(* CODESYS project CintasSoplado.project
   Title: CintasSoplado
   Version: 0.0.0.0
   Author: serbogr1

Project tree, tasks and I/O mapping:
  MyController : TM241CE40R, Schneider Electric, order no. TM241CE40R, version 4.0.6.18
    application Application
      libraries: Toolbox, 2.2.0.0 (Schneider Electric)
      task MAST (cyclic, interval 50 ms, priority 15, watchdog 100 ms x 1) calls ProcesoUno, ProcesoDos, Pulsadores, PID
      global variables GVL
      visualisation HMIW_Control
      image pool ImagePool
      program ProcesoDos [SFC]: E2_active, E8_active
      program ProcesoUno [SFC]: E8_active, E7_active, E9_active, E10_active, E11_active, E12_active
      program Pulsadores [LD]
      program PruebaAnalogica [ST]
      program PID [LD]
    DI : Digital Inputs, Schneider Electric, version 4.0.6.18
        input  idwDI_IDW0 : DWORD  // IDW0
        input  ibDI_IB1 : BYTE  // IB1
    DQ : Digital Outputs, Schneider Electric, version 4.0.6.18
        output qwDQ_QW0 : WORD  // QW0
        output qbDQ_QB1 : BYTE  // QB1
    Counters : Counters, Schneider Electric, version 4.0.6.18
    Pulse_Generators : Pulse Generators, Schneider Electric, version 4.0.6.18
    Cartridge_1 : Cartridge, Schneider Electric, version 4.0.6.18
      TMC4AI2 : TMC4AI2, Schneider Electric, order no. TMC4AI2, version 1.0.1.0
          input  iiTMC4AI2_IW0 : INT  // IW0
          input  iiTMC4AI2_IW1 : INT  // IW1
          input  ibTMC4AI2_IW2 : BYTE  // IW2
    Cartridge_2 : Cartridge, Schneider Electric, version 4.0.6.18
      TMC4AQ2 : TMC4AQ2, Schneider Electric, order no. TMC4AQ2, version 1.0.1.1
          output qiTMC4AQ2_QW0 : INT  // QW0
          output qiTMC4AQ2_QW1 : INT  // QW1
          input  ibTMC4AQ2_IW0 : BYTE  // IW0
    IO_Bus : IO bus - TM3, Schneider Electric, version 4.0.6.18
    COM_Bus : COM bus, Schneider Electric, version 4.0.6.18
    Ethernet_1 : Ethernet Network, Schneider Electric, version 4.0.6.18
        settings: WebServer = TRUE; FTP Server = TRUE; SoMachine Protocol = TRUE; Modbus Server = TRUE; NetManage Protocol = TRUE; SNMP protocol = TRUE; Enable Routing = FALSE; WebVisu protocol = TRUE; DHCP Server Active = FALSE
    Serial_Line_1 : Serial line, Schneider Electric, version 4.0.6.18
      SoMachine_Network_Manager : SoMachine-Network Manager, Schneider Electric, version 4.0.0.2
    Serial_Line_2 : Serial line, Schneider Electric, version 4.0.6.18
      Modbus_Manager : Modbus Manager, Schneider Electric, version 4.0.0.2
  text list GlobalTextList
*)

// MyController/Application/GVL
VAR_GLOBAL
END_VAR

// MyController/Application/ProcesoUno
PROGRAM ProcesoUno
VAR
	bS_FC_Empujador_1          AT %IX0.0: BOOL; (*I1*)
	bS_IC_Empujador_1          AT %IX0.1: BOOL; (*I2*)
	bS_FC_Empujador_2          AT %IX0.2: BOOL; (*I3*)
	bS_IC_Empujador_2          AT %IX0.3: BOOL; (*I4*)
	bS_FT_Empujador_1          AT %IX0.4: BOOL; (*I5*)
	bS_FT_Fresadora            AT %IX0.5: BOOL; (*I6*)
	bS_FT_Carga                AT %IX0.6: BOOL; (*I7*)
	bS_FT_Taladro              AT %IX0.7: BOOL; (*I8*)
	bS_FT_Salida               AT %IX1.0: BOOL; (*I9*)
	
	bA_M_Cinta_Alimentacion    AT %QX1.0: BOOL; (*Q5*)
	bA_M_Cinta_Fresadora       AT %QX1.1: BOOL; (*Q6*)
	bA_M_Fresadora             AT %QX1.2: BOOL; (*Q7*)
	bA_M_Cinta_Taladro         AT %QX1.3: BOOL; (*Q8*)
	bA_M_Taladro               AT %QX1.4: BOOL; (*Q9*)
	bA_M_Cinta_Salida          AT %QX1.5: BOOL; (*Q10*)
	bA_Habilitar_Sistema       AT %QX1.6: BOOL; (*Q11*)
	
	bBotonEmergenciaHMI        AT %MX0.0: BOOL; (*Boton Emergencia HMI*)
	bBotonEmergenciaHMIW       AT %MX0.2: BOOL; (*Boton Emergencia HMIW*)	
	bBotonInicioHMI            AT %MX0.1: BOOL; (*Boton Inicio HMI*)
	bBotonInicioHMIW           AT %MX0.3: BOOL; (*Boton Inicio HMIW*)
    bBotonPiezaHMIW            AT %MX1.7: BOOL; (*Boton Poner Pieza*)
    bSiguientePieza            AT %MX0.4: BOOL; (*Activa cuando se puede poner la siguiente pieza*)	
	bFinSoplado                         : BOOL; (*Activa Cuando termina Soplado*)
	iTiempoFresado                      : LINT:=1;
	iTiempoTaladrado                    : LINT:=1;
	iTiempoSoplado                      : LINT:=1;	

END_VAR

VAR_OUTPUT
	tEmpujador_1   : TIME:=T#1S;
	tFresado       : TIME:=T#1S;
	(*tTaladrado     : TIME:=T#1S;*)
	tEmpujador_2   : TIME:=T#1S;
END_VAR

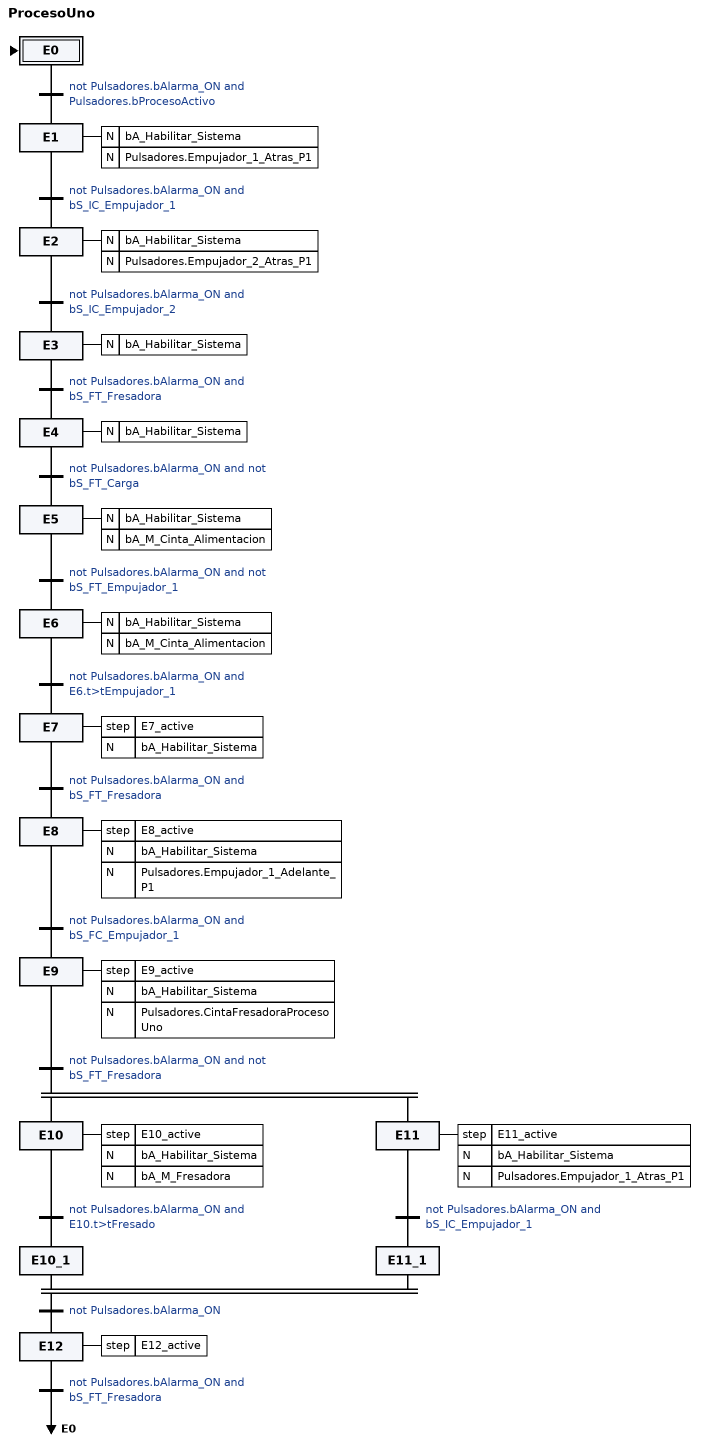
INITIAL_STEP E0:
END_STEP
TRANSITION FROM E0 TO E1
    := not Pulsadores.bAlarma_ON and Pulsadores.bProcesoActivo;
END_TRANSITION
STEP E1:
    bA_Habilitar_Sistema(N);
    Pulsadores.Empujador_1_Atras_P1(N);
END_STEP
TRANSITION FROM E1 TO E2
    := not Pulsadores.bAlarma_ON and bS_IC_Empujador_1;
END_TRANSITION
STEP E2:
    bA_Habilitar_Sistema(N);
    Pulsadores.Empujador_2_Atras_P1(N);
END_STEP
TRANSITION FROM E2 TO E3
    := not Pulsadores.bAlarma_ON and bS_IC_Empujador_2;
END_TRANSITION
STEP E3:
    bA_Habilitar_Sistema(N);
END_STEP
TRANSITION FROM E3 TO E4
    := not Pulsadores.bAlarma_ON and bS_FT_Fresadora;
END_TRANSITION
STEP E4:
    bA_Habilitar_Sistema(N);
END_STEP
TRANSITION FROM E4 TO E5
    := not Pulsadores.bAlarma_ON and not bS_FT_Carga;
END_TRANSITION
STEP E5:
    bA_Habilitar_Sistema(N);
    bA_M_Cinta_Alimentacion(N);
END_STEP
TRANSITION FROM E5 TO E6
    := not Pulsadores.bAlarma_ON and not bS_FT_Empujador_1;
END_TRANSITION
STEP E6:
    bA_Habilitar_Sistema(N);
    bA_M_Cinta_Alimentacion(N);
END_STEP
TRANSITION FROM E6 TO E7
    := not Pulsadores.bAlarma_ON and E6.t>tEmpujador_1;
END_TRANSITION
STEP E7:
    E7_active(N);  // step action
    bA_Habilitar_Sistema(N);
END_STEP
TRANSITION FROM E7 TO E8
    := not Pulsadores.bAlarma_ON and bS_FT_Fresadora;
END_TRANSITION
STEP E8:
    E8_active(N);  // step action
    bA_Habilitar_Sistema(N);
    Pulsadores.Empujador_1_Adelante_P1(N);
END_STEP
TRANSITION FROM E8 TO E9
    := not Pulsadores.bAlarma_ON and bS_FC_Empujador_1;
END_TRANSITION
STEP E9:
    E9_active(N);  // step action
    bA_Habilitar_Sistema(N);
    Pulsadores.CintaFresadoraProcesoUno(N);
END_STEP
TRANSITION FROM E9 TO (E10, E11)
    := not Pulsadores.bAlarma_ON and not bS_FT_Fresadora;
END_TRANSITION
STEP E10:
    E10_active(N);  // step action
    bA_Habilitar_Sistema(N);
    bA_M_Fresadora(N);
END_STEP
TRANSITION FROM E10 TO E10_1
    := not Pulsadores.bAlarma_ON and E10.t>tFresado;
END_TRANSITION
STEP E10_1:
END_STEP
STEP E11:
    E11_active(N);  // step action
    bA_Habilitar_Sistema(N);
    Pulsadores.Empujador_1_Atras_P1(N);
END_STEP
TRANSITION FROM E11 TO E11_1
    := not Pulsadores.bAlarma_ON and bS_IC_Empujador_1;
END_TRANSITION
STEP E11_1:
END_STEP
TRANSITION FROM (E10_1, E11_1) TO E12
    := not Pulsadores.bAlarma_ON;
END_TRANSITION
STEP E12:
    E12_active(N);  // step action
END_STEP
TRANSITION FROM E12 TO E0
    := not Pulsadores.bAlarma_ON and bS_FT_Fresadora;
END_TRANSITION

ACTION E8_active:
IF bS_FT_Carga THEN
	bSiguientePieza := TRUE;
ELSIF NOT bS_FT_Carga THEN
	bSiguientePieza := FALSE;
END_IF
END_ACTION

ACTION E7_active:
IF bS_FT_Carga THEN
	bSiguientePieza := TRUE;
ELSIF NOT bS_FT_Carga THEN
	bSiguientePieza := FALSE;
END_IF
END_ACTION

ACTION E9_active:
IF bS_FT_Carga THEN
	bSiguientePieza := TRUE;
ELSIF NOT bS_FT_Carga THEN
	bSiguientePieza := FALSE;
END_IF
END_ACTION

ACTION E10_active:
IF bS_FT_Carga THEN
	bSiguientePieza := TRUE;
ELSIF NOT bS_FT_Carga THEN
	bSiguientePieza := FALSE;
END_IF

    tFresado := LINT_TO_TIME(iTiempoFresado*1000);
END_ACTION

ACTION E11_active:
IF bS_FT_Carga THEN
	bSiguientePieza := TRUE;
ELSIF NOT bS_FT_Carga THEN
	bSiguientePieza := FALSE;
END_IF
END_ACTION

ACTION E12_active:
IF bS_FT_Carga THEN
	bSiguientePieza := TRUE;
ELSIF NOT bS_FT_Carga THEN
	bSiguientePieza := FALSE;
END_IF
END_ACTION

END_PROGRAM

// MyController/Application/ProcesoDos
PROGRAM ProcesoDos
VAR
		tTaladrado        : TIME:=T#1S;
		rPiezasTerminadas : INT:=0;
END_VAR

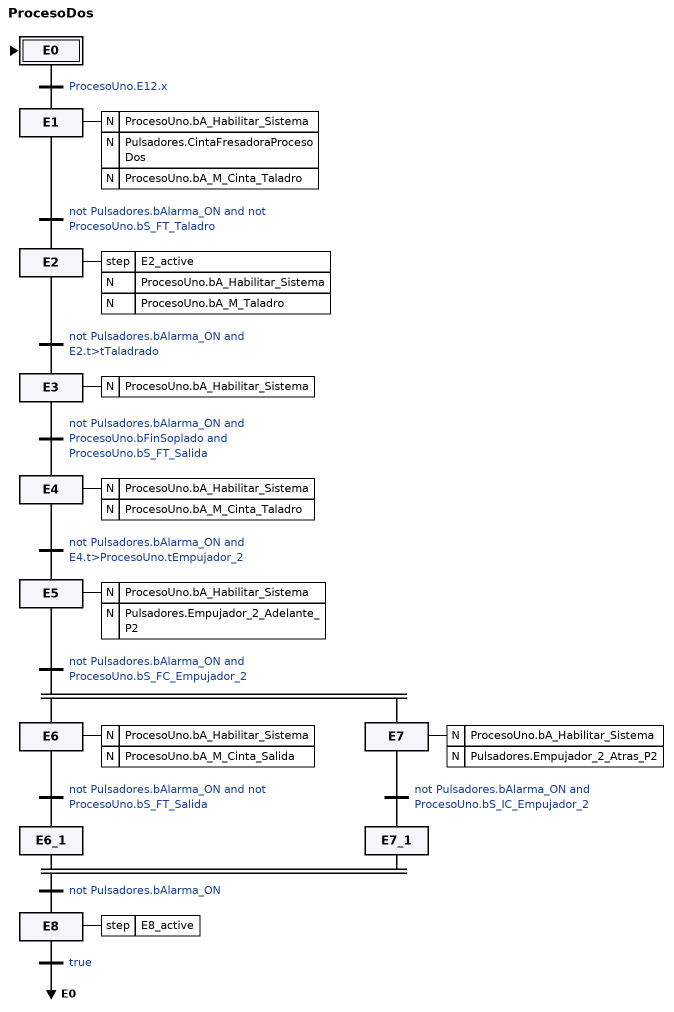
INITIAL_STEP E0:
END_STEP
TRANSITION FROM E0 TO E1
    := ProcesoUno.E12.x;
END_TRANSITION
STEP E1:
    ProcesoUno.bA_Habilitar_Sistema(N);
    Pulsadores.CintaFresadoraProcesoDos(N);
    ProcesoUno.bA_M_Cinta_Taladro(N);
END_STEP
TRANSITION FROM E1 TO E2
    := not Pulsadores.bAlarma_ON and not ProcesoUno.bS_FT_Taladro;
END_TRANSITION
STEP E2:
    E2_active(N);  // step action
    ProcesoUno.bA_Habilitar_Sistema(N);
    ProcesoUno.bA_M_Taladro(N);
END_STEP
TRANSITION FROM E2 TO E3
    := not Pulsadores.bAlarma_ON and E2.t>tTaladrado;
END_TRANSITION
STEP E3:
    ProcesoUno.bA_Habilitar_Sistema(N);
END_STEP
TRANSITION FROM E3 TO E4
    := not Pulsadores.bAlarma_ON and ProcesoUno.bFinSoplado and ProcesoUno.bS_FT_Salida;
END_TRANSITION
STEP E4:
    ProcesoUno.bA_Habilitar_Sistema(N);
    ProcesoUno.bA_M_Cinta_Taladro(N);
END_STEP
TRANSITION FROM E4 TO E5
    := not Pulsadores.bAlarma_ON and E4.t>ProcesoUno.tEmpujador_2;
END_TRANSITION
STEP E5:
    ProcesoUno.bA_Habilitar_Sistema(N);
    Pulsadores.Empujador_2_Adelante_P2(N);
END_STEP
TRANSITION FROM E5 TO (E6, E7)
    := not Pulsadores.bAlarma_ON and ProcesoUno.bS_FC_Empujador_2;
END_TRANSITION
STEP E6:
    ProcesoUno.bA_Habilitar_Sistema(N);
    ProcesoUno.bA_M_Cinta_Salida(N);
END_STEP
TRANSITION FROM E6 TO E6_1
    := not Pulsadores.bAlarma_ON and not ProcesoUno.bS_FT_Salida;
END_TRANSITION
STEP E6_1:
END_STEP
STEP E7:
    ProcesoUno.bA_Habilitar_Sistema(N);
    Pulsadores.Empujador_2_Atras_P2(N);
END_STEP
TRANSITION FROM E7 TO E7_1
    := not Pulsadores.bAlarma_ON and ProcesoUno.bS_IC_Empujador_2;
END_TRANSITION
STEP E7_1:
END_STEP
TRANSITION FROM (E6_1, E7_1) TO E8
    := not Pulsadores.bAlarma_ON;
END_TRANSITION
STEP E8:
    E8_active(N);  // step action
END_STEP
TRANSITION FROM E8 TO E0
    := true;
END_TRANSITION

ACTION E2_active:
  
tTaladrado := LINT_TO_TIME(ProcesoUno.iTiempoTaladrado*1000);
END_ACTION

ACTION E8_active:
IF NOT ProcesoUno.bS_FT_Salida THEN
	rPiezasTerminadas := rPiezasTerminadas + 1;
END_IF
END_ACTION

END_PROGRAM

// MyController/Application/Pulsadores
PROGRAM Pulsadores
VAR
	bA_M_Empujador_1_Adelante  AT %QX0.4: BOOL; (*Q1*)
	bA_M_Empujador_1_Atras     AT %QX0.5: BOOL; (*Q2*)
	bA_M_Empujador_2_Adelante  AT %QX0.6: BOOL; (*Q3*)
	bA_M_Empujador_2_Atras     AT %QX0.7: BOOL; (*Q4*)	

	bAlarma_ON                  :BOOL; (*Activa cuando se pulsa alarma*)
	bProcesoActivo              :BOOL;	(*Activa cuando se pulsa inicio*)	
	CintaFresadoraProcesoUno    :BOOL;
	CintaFresadoraProcesoDos    :BOOL;
	Empujador_1_Adelante_P1     :BOOL;
	Empujador_1_Adelante_P2     :BOOL;
	Empujador_2_Adelante_P1     :BOOL;	
    Empujador_2_Adelante_P2     :BOOL;
	Empujador_1_Atras_P1        :BOOL;
	Empujador_1_Atras_P2        :BOOL;	
	Empujador_2_Atras_P1        :BOOL;
	Empujador_2_Atras_P2        :BOOL;		
	rLongTime: INT;
END_VAR

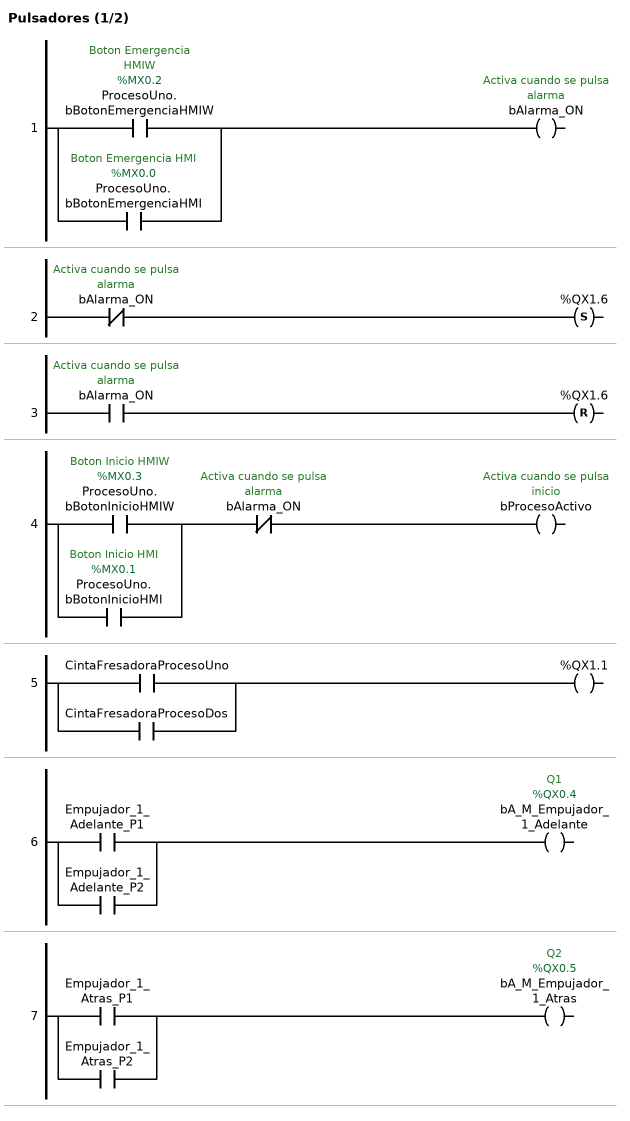
// NETWORK 1
//   ProcesoUno.bBotonEmergenciaHMIW: Boton Emergencia HMIW | AT %MX0.2
//   ProcesoUno.bBotonEmergenciaHMI: Boton Emergencia HMI | AT %MX0.0
//   bAlarma_ON: Activa cuando se pulsa alarma
bAlarma_ON := ProcesoUno.bBotonEmergenciaHMIW OR ProcesoUno.bBotonEmergenciaHMI;

// NETWORK 2
//   bAlarma_ON: Activa cuando se pulsa alarma
%QX1.6 S= NOT bAlarma_ON;

// NETWORK 3
//   bAlarma_ON: Activa cuando se pulsa alarma
%QX1.6 R= bAlarma_ON;

// NETWORK 4
//   ProcesoUno.bBotonInicioHMIW: Boton Inicio HMIW | AT %MX0.3
//   ProcesoUno.bBotonInicioHMI: Boton Inicio HMI | AT %MX0.1
//   bAlarma_ON: Activa cuando se pulsa alarma
//   bProcesoActivo: Activa cuando se pulsa inicio
bProcesoActivo := (ProcesoUno.bBotonInicioHMIW OR ProcesoUno.bBotonInicioHMI) AND NOT bAlarma_ON;

// NETWORK 5
%QX1.1 := CintaFresadoraProcesoUno OR CintaFresadoraProcesoDos;

// NETWORK 6
//   bA_M_Empujador_1_Adelante: Q1 | AT %QX0.4
bA_M_Empujador_1_Adelante := Empujador_1_Adelante_P1 OR Empujador_1_Adelante_P2;

// NETWORK 7
//   bA_M_Empujador_1_Atras: Q2 | AT %QX0.5
bA_M_Empujador_1_Atras := Empujador_1_Atras_P1 OR Empujador_1_Atras_P2;

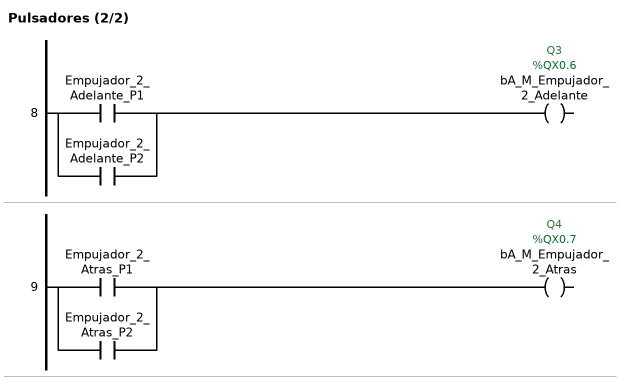
// NETWORK 8
//   bA_M_Empujador_2_Adelante: Q3 | AT %QX0.6
bA_M_Empujador_2_Adelante := Empujador_2_Adelante_P1 OR Empujador_2_Adelante_P2;

// NETWORK 9
//   bA_M_Empujador_2_Atras: Q4 | AT %QX0.7
bA_M_Empujador_2_Atras := Empujador_2_Atras_P1 OR Empujador_2_Atras_P2;

END_PROGRAM

// MyController/Application/PID
PROGRAM PID
VAR
	vActuador        AT %QW2 : WORD;
	rActuador                : REAL;
	vSensor          AT %IW3 : WORD;	
	voltsSensorSim           : WORD:=2500;
	rSensor                  : REAL;	
	rReferencia              : REAL:=-26;
	AutoManual               : BOOL;
	ResetPID                 : BOOL;
	FB_Scaling_vS            : FB_Scaling; (*Escalado para tensión del sensor*)
	FB_Scaling_vA            : FB_Scaling; (*Escalado para tensión al actuador*)
	PID_ControHelice         : Util.PID;

END_VAR

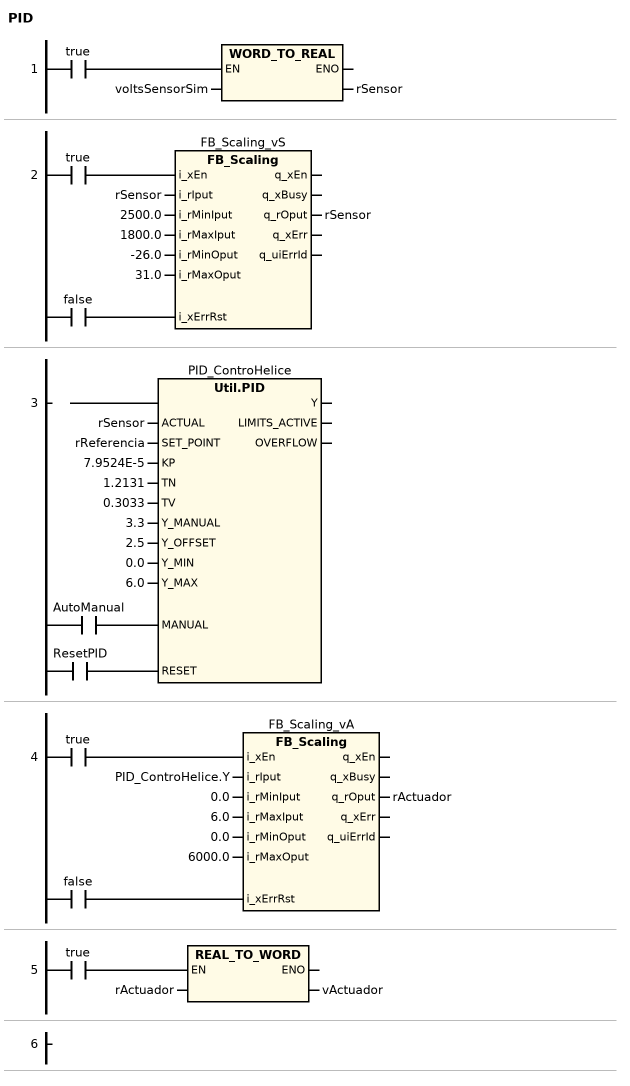
// NETWORK 1
IF true THEN rSensor := WORD_TO_REAL(voltsSensorSim); END_IF

// NETWORK 2
//   FB_Scaling_vS: Escalado para tensión del sensor
FB_Scaling_vS(
    i_xEn := true,
    i_rIput := rSensor,
    i_rMinIput := 2500.0,
    i_rMaxIput := 1800.0,
    i_rMinOput := -26.0,
    i_rMaxOput := 31.0,
    i_xErrRst := false,
    q_rOput => rSensor); // FB_Scaling

// NETWORK 3
PID_ControHelice(
    ACTUAL := rSensor,
    SET_POINT := rReferencia,
    KP := 7.9524E-5,
    TN := 1.2131,
    TV := 0.3033,
    Y_MANUAL := 3.3,
    Y_OFFSET := 2.5,
    Y_MIN := 0.0,
    Y_MAX := 6.0,
    MANUAL := AutoManual,
    RESET := ResetPID); // Util.PID

// NETWORK 4
//   FB_Scaling_vA: Escalado para tensión al actuador
//   PID_ControHelice.Y: manipulated variable, set value
FB_Scaling_vA(
    i_xEn := true,
    i_rIput := PID_ControHelice.Y,
    i_rMinIput := 0.0,
    i_rMaxIput := 6.0,
    i_rMinOput := 0.0,
    i_rMaxOput := 6000.0,
    i_xErrRst := false,
    q_rOput => rActuador); // FB_Scaling

// NETWORK 5
//   vActuador: AT %QW2
IF true THEN vActuador := REAL_TO_WORD(rActuador); END_IF

// NETWORK 6

END_PROGRAM

// MyController/Application/PruebaAnalogica
PROGRAM PruebaAnalogica
VAR
	tensionSalida: WORD;
	tensionEntrada: WORD;	
END_VAR


%QW2 := tensionSalida;
tensionEntrada := %IW3;

END_PROGRAM

// MyController/Application/HMIW_Control
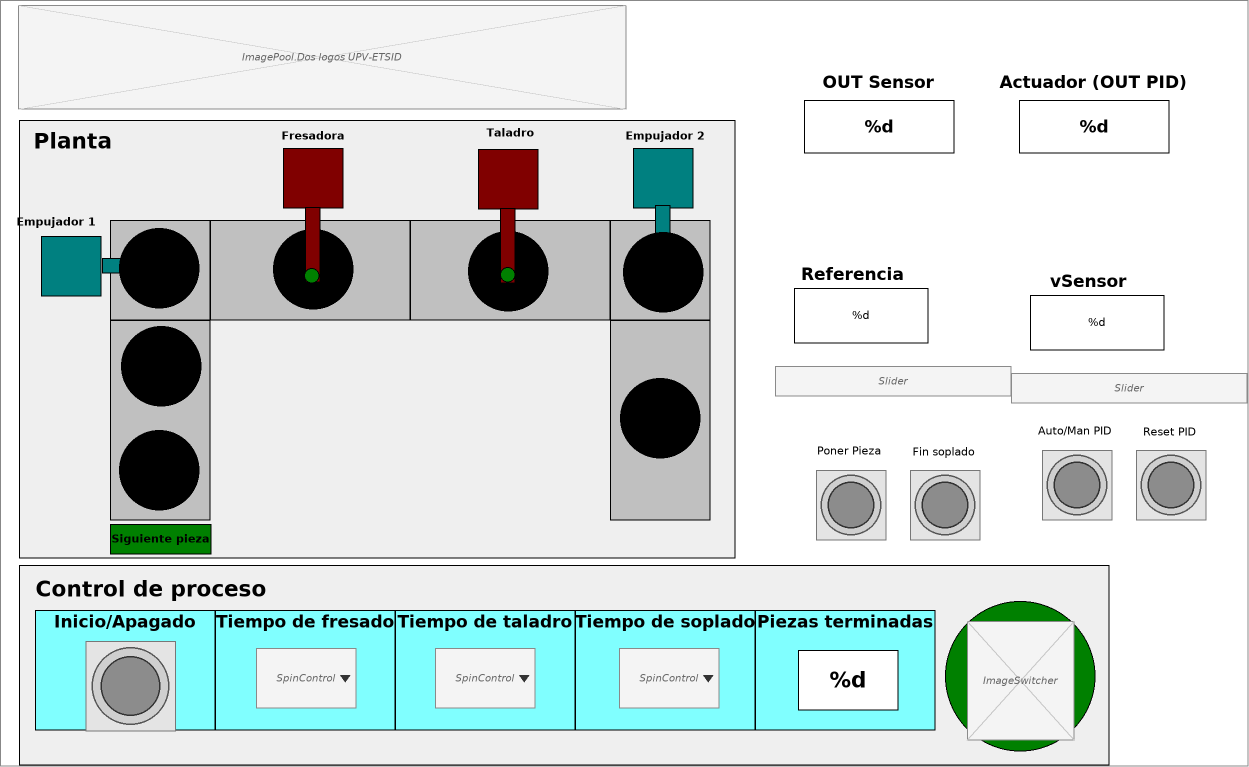
VISUALIZATION HMIW_Control  // 1249x767
    Rectangle (19,565 1090x200)
    Rectangle (19,120 716x438)
    Rectangle (110,220 100x100)
    Rectangle (110,320 100x200)
    Rectangle (610,320 100x200)
    Rectangle (610,220 100x100)
    Rectangle (210,220 200x100)
    Rectangle (410,220 200x100)
    Rectangle (35,610 180x120), "Inicio/Apagado"
    Rectangle (215,610 180x120), "Tiempo de fresado"
    Rectangle (395,610 180x120), "Tiempo de taladro"
    Rectangle (575,610 180x120), "Tiempo de soplado"
    Rectangle (755,610 180x120), "Piezas terminadas"
    Label (40,574 222x30), "Control de proceso"
    Label (809,436 80x30), "Poner Pieza"
    PushSwitch (816,470 70x70), variable: ProcesoUno.bBotonPiezaHMIW, behaviour: TAP, style: Switch-PushSwitch-Gray
    PushSwitch (910,470 70x70), variable: ProcesoUno.bFinSoplado, behaviour: TAP, style: Switch-PushSwitch-Gray
    Label (904,437 79x30), "Fin soplado"
    Label (789,259 127x30), "Referencia"
    SpinControl (256,648 100x60), variable: ProcesoUno.iTiempoFresado
    SpinControl (435,648 100x60), variable: ProcesoUno.iTiempoTaladrado
    SpinControl (619,648 100x60), variable: ProcesoUno.iTiempoSoplado
    PushSwitchLed (85,641 91x90), variable: ProcesoUno.bBotonInicioHMIW, behaviour: TOGGLE, style: Switch-PushSwitchLed-Gray
    Ellipse (119,430 80x80), invisible if: ProcesoUno.bS_FT_Carga
    Ellipse (121,326 80x80), invisible if: ProcesoUno.bS_FT_Empujador_1
    Ellipse (273,229 80x80), invisible if: ProcesoUno.bS_FT_Fresadora
    Ellipse (468,231 80x80), invisible if: ProcesoUno.bS_FT_Taladro
    Ellipse (620,378 80x80), invisible if: ProcesoUno.bS_FT_Salida
    RoundedRectangle (798,650 100x60), "%d", text variable: ProcesoDos.rPiezasTerminadas
    RoundedRectangle (41,236 60x60)
    RoundedRectangle (633,148 60x60)
    RoundedRectangle (283,148 60x60)
    RoundedRectangle (478,149 60x60)
    Rectangle (305,207 15x75)
    Rectangle (500,208 15x75)
    Rectangle (655,205 15x75), invisible if: not ProcesoUno.bA_M_Empujador_2_Adelante
    Ellipse (304,268 15x15), colour toggle: ProcesoUno.bA_M_Fresadora
    Ellipse (500,267 15x15), colour toggle: ProcesoUno.bA_M_Taladro
    Rectangle (102,258 75x15), invisible if: not ProcesoUno.bA_M_Empujador_1_Adelante
    Ellipse (623,232 80x80), invisible if: ProcesoUno.bS_IC_Empujador_2
    Ellipse (119,228 80x80), invisible if: ProcesoUno.bS_IC_Empujador_1
    Label (277,121 72x30), "Fresadora"
    Label (15,207 82x30), "Empujador 1"
    Label (475,118 71x30), "Taladro"
    Label (629,121 72x30), "Empujador 2"
    Image (18,5 608x104), image: ImagePool.Dos logos UPV-ETSID
    Label (27,127 92x28), "Planta"
    Ellipse (945,601 150x150), colour toggle: ProcesoUno.bBotonEmergenciaHMIW
    ImageSwitcher (967,621 107x119), variable: ProcesoUno.bBotonEmergenciaHMIW, background image: ImagePool.BotonEmergencia, image: ImagePool.BotonEmergencia, behaviour: TOGGLE
    Rectangle (1019,100 150x53), "%d", text variable: PID.vActuador
    Label (999,67 189x30), "Actuador (OUT PID)"
    RoundedRectangle (110,524 101x30), "Siguiente pieza", colour toggle: ProcesoUno.bSiguientePieza
    Rectangle (804,100 150x53), "%d", text variable: PID.vSensor
    Label (784,67 189x30), "OUT Sensor"
    Slider (775,366 236x30), variable: PID.rReferencia, scale -26..31
    RoundedRectangle (794,288 134x55), "%d", text variable: PID.rReferencia
    Label (1025,266 127x30), "vSensor"
    Slider (1011,373 236x30), variable: PID.voltsSensorSim, scale 1800..2500
    RoundedRectangle (1030,295 134x55), "%d", text variable: PID.voltsSensorSim
    Label (1035,416 80x30), "Auto/Man PID"
    PushSwitch (1042,450 70x70), variable: PID.AutoManual, behaviour: TOGGLE, style: Switch-PushSwitch-Gray
    PushSwitch (1136,450 70x70), variable: PID.ResetPID, behaviour: TAP, style: Switch-PushSwitch-Gray
    Label (1130,417 79x30), "Reset PID"
END_VISUALIZATION
